TYPE InputBase_8311D824 :
STRUCT
END_STRUCT
END_TYPE

(* stored: Version 1.2.0.0, ProductVersion 3.1.4024.9
   DUT InputBase_8311D824: Id {7d28777f-077e-4502-8987-eced6970db81} *)
